Staubli VAL3: GetPostion.dtx

bool bOver
jointRx j1 = {j1=1.78216, j2=38.861437, j3=114.367622}
jointRx jNow = {j1=26.247439, j2=37.206969, j3=118.159168, j4=-90.166827, j5=10.750799, j6=112.277964}
mdesc mMdesc
mdesc mNomSpeed
pointRx p1 = {x=544.540194, y=303.457147, z=-190.997145, rx=0.899428, ry=153.242342, rz=-1.996136, fatherId=world[0]}
pointRx pNow = {x=544.540194, y=303.457147, z=-190.997145, rx=0.899428, ry=153.242342, rz=-1.996136, shoulder=lefty, elbow=epositive, wrist=wpositive, fatherId=world[0]}
tool tTool = {fatherId=flange[0], ioLink=valve1}
num nFileID
num nJointForce[6]
num nForceData[1000 6]
